// TIA Portal V16 export
// export: Created 2021-09-08T12:46:09.8350938Z, ExportSetting WithDefaults, DisplayName Totally Integrated Automation Portal, DisplayVersion V16 Update 3, DisplayName TIA Portal Version Control Interface, DisplayVersion V16 Update 2, DisplayName TIA Portal Openness, DisplayVersion V16 Update 3, DisplayName TIA Portal Teamcenter Gateway, DisplayVersion V16, DisplayName STEP 7 Professional, DisplayVersion V16 Update 3, DisplayName STEP 7 Safety, DisplayVersion V16, DisplayName WinCC Advanced, DisplayVersion V16 Update 3
FUNCTION_BLOCK "AvCntrl"   // FB81, LAD
{ S7_Optimized_Access := 'FALSE' }
VERSION : 0.1
// #ST:
// 0 0 - закрыта - стоп 
// 1 1- открыта - работа
// 2 2 -открывается - запускается
// 3 4 -закрывается - останавливается 
// 4 8 - ошибка питания
// 5 16 - ошибка концевиков - закрытия
// 6 32 - Блокировка
// 7 64 - сборная авария
// 8 128 - ошибка концевиков - открытия
// 9 256 - не выбран режим
// 10 - 512 - показывать кнопки ручного управления
// 
// БИТ 13 - РЕЖИМ
// бит 14 - состояние концевиков - открыто
// 15 - закрыто
// stored: AutoNumber false, IsIECCheckEnabled true, SetENOAutomatically false, UDAEnableTagReadback false
   VAR_INPUT
      power : Bool;   // питание устройства
      open : Bool;   // Задвижка открыта
      close : Bool;   // Задвижка закрыта
   END_VAR
   VAR_OUTPUT
      qKm : Bool;   // Выход на управление механизмом 0-стоп, 1-пуск
   END_VAR
   VAR_IN_OUT
      dev : "Av";
   END_VAR
   VAR DB_SPECIFIC
      Ack : Bool;   // Сброс Аварий
      ErrorOC : Bool;   // Признак аварии по закрытию или открытию
      ErrorPower : Bool;   // Признак аварии питания
      ErrorDis : Bool;   // Признак внешней блокировки
      Error : Bool;   // Признак наличия сборной ошибки
      qON : Bool;   // Выход для управления механизмом
      closed : Bool;
      opened : Bool;
      closing : Bool;
      opening : Bool;
      errOpen : Bool;
      errClose : Bool;
      timerOpening { S7_SetPoint := 'True'} : TON_TIME;
      timerClosing { S7_SetPoint := 'True'} : TON_TIME;
      tClose : Time;
      tOpen : Time;
   END_VAR
   VAR
      AvAckAlarm_Instance { S7_SetPoint := 'True'} : "AvAckAlarm";
   END_VAR
   VAR_TEMP
      tmpDInt : DInt;
   END_VAR
   VAR_TEMP   // added for the SCL form of the ladder/FBD networks
      _w1 : Bool;
   END_VAR
BEGIN

REGION Network 1: Сброс состояния
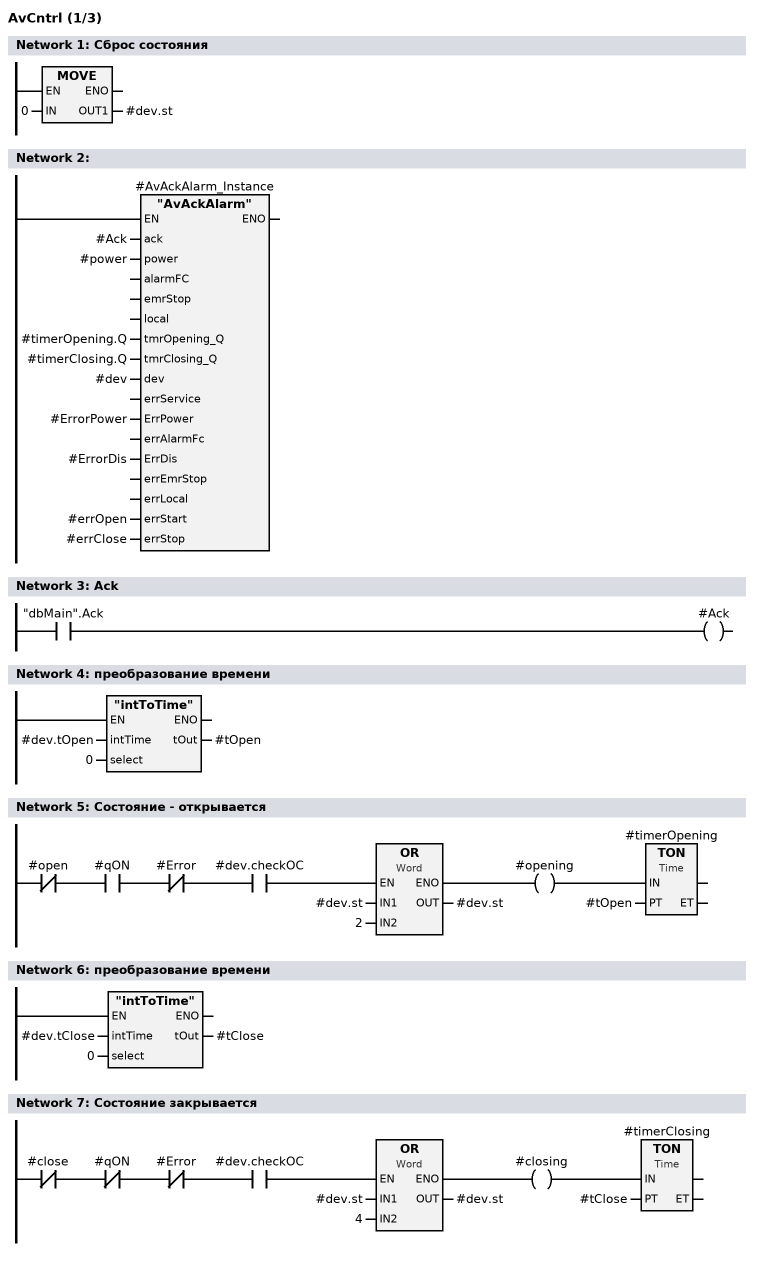
   RUNG wire#powerrail
      { S7_GenerateENO := "TRUE" } Move(in := 0, out1 => #dev.st)
   END_RUNG
   // the same network as SCL:
   #dev.st := 0;
END_REGION

REGION Network 2
   RUNG wire#powerrail
      #AvAckAlarm_Instance(ack := #Ack, power := #power, alarmFC :=, emrStop :=, local :=, tmrOpening_Q := #timerOpening.Q, tmrClosing_Q := #timerClosing.Q, dev := #dev, errService :=, ErrPower := #ErrorPower, errAlarmFc :=, ErrDis := #ErrorDis, errEmrStop :=, errLocal :=, errStart := #errOpen, errStop := #errClose)
   END_RUNG
   // the same network as SCL:
   #AvAckAlarm_Instance(ack := #Ack,   // "AvAckAlarm"
                        power := #power,
                        tmrOpening_Q := #timerOpening.Q,
                        tmrClosing_Q := #timerClosing.Q,
                        dev := #dev,
                        ErrPower := #ErrorPower,
                        ErrDis := #ErrorDis,
                        errStart := #errOpen,
                        errStop := #errClose);
END_REGION

REGION Network 3: Ack
   RUNG wire#powerrail
      Contact( "dbMain".Ack )
      Coil( #Ack )
   END_RUNG
   // the same network as SCL:
   #Ack := "dbMain".Ack;
END_REGION

REGION Network 4: преобразование времени
   RUNG wire#powerrail
      "intToTime"(intTime := #dev.tOpen, select := 0, tOut => #tOpen)
   END_RUNG
   // the same network as SCL:
   "intToTime"(intTime := #dev.tOpen, select := 0, tOut => #tOpen);
END_REGION

REGION Network 5: Состояние - открывается
   #_w1 := NOT #open AND #qON AND NOT #Error AND #dev.checkOC;
   IF #_w1 THEN #dev.st := #dev.st OR 2; END_IF;
   #opening := #_w1;
   #timerOpening(IN := #_w1, PT := #tOpen);   // TON
END_REGION

REGION Network 6: преобразование времени
   RUNG wire#powerrail
      "intToTime"(intTime := #dev.tClose, select := 0, tOut => #tClose)
   END_RUNG
   // the same network as SCL:
   "intToTime"(intTime := #dev.tClose, select := 0, tOut => #tClose);
END_REGION

REGION Network 7: Состояние закрывается
   #_w1 := NOT #close AND NOT #qON AND NOT #Error AND #dev.checkOC;
   IF #_w1 THEN #dev.st := #dev.st OR 4; END_IF;
   #closing := #_w1;
   #timerClosing(IN := #_w1, PT := #tClose);   // TON
END_REGION

REGION Network 8: Признак аварии по закрытию или открытию
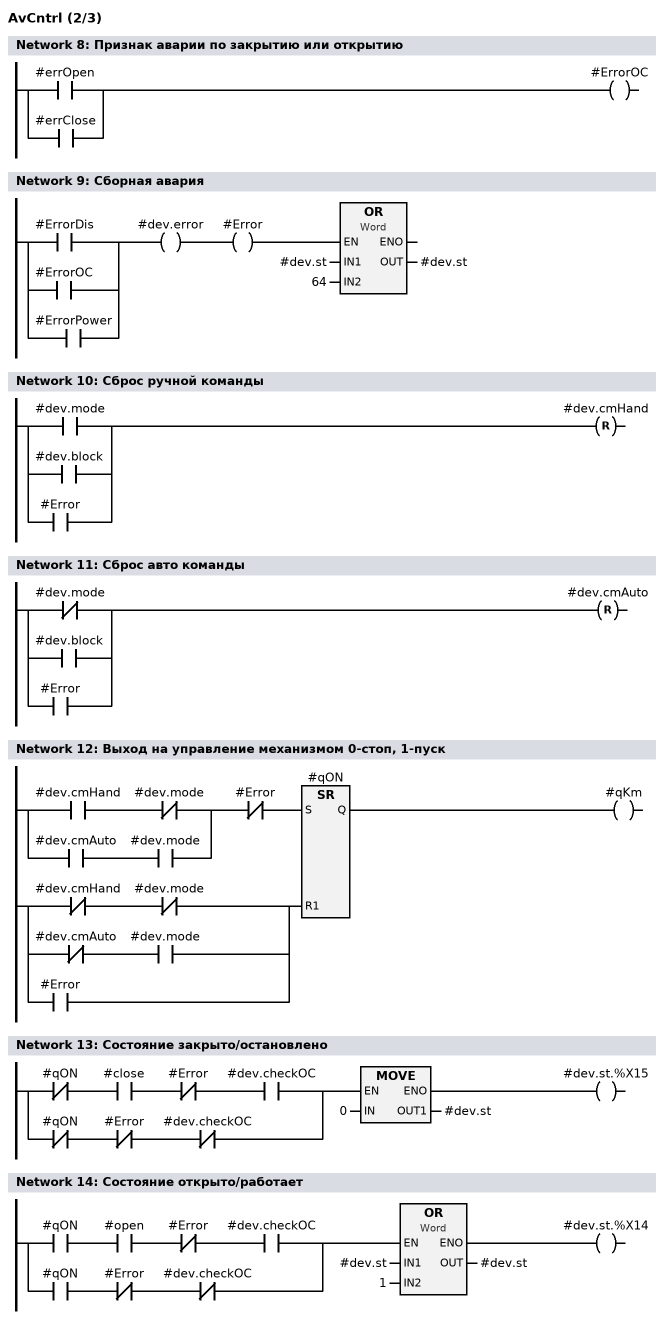
   RUNG wire#powerrail
      Contact( #errOpen )
      wire#w1
      Coil( #ErrorOC )
   END_RUNG
   RUNG wire#powerrail
      Contact( #errClose )
   END_RUNG wire#w1
   // the same network as SCL:
   #ErrorOC := #errOpen OR #errClose;
END_REGION

REGION Network 9: Сборная авария
   #dev.error := #ErrorDis OR #ErrorOC OR #ErrorPower;
   #Error := #dev.error;
   IF #dev.error THEN #dev.st := #dev.st OR 64; END_IF;
END_REGION

REGION Network 10: Сброс ручной команды
   RUNG wire#powerrail
      Contact( #dev.mode )
      wire#w1
      R_Coil( #dev.cmHand )
   END_RUNG
   RUNG wire#powerrail
      Contact( #dev.block )
   END_RUNG wire#w1
   RUNG wire#powerrail
      Contact( #Error )
   END_RUNG wire#w1
   // the same network as SCL:
   IF #dev.mode OR #dev.block OR #Error THEN #dev.cmHand := FALSE; END_IF;
END_REGION

REGION Network 11: Сброс авто команды
   RUNG wire#powerrail
      I_Contact( #dev.mode )
      wire#w1
      R_Coil( #dev.cmAuto )
   END_RUNG
   RUNG wire#powerrail
      Contact( #dev.block )
   END_RUNG wire#w1
   RUNG wire#powerrail
      Contact( #Error )
   END_RUNG wire#w1
   // the same network as SCL:
   IF NOT #dev.mode OR #dev.block OR #Error THEN #dev.cmAuto := FALSE; END_IF;
END_REGION

REGION Network 12: Выход на управление механизмом 0-стоп, 1-пуск
   RUNG wire#powerrail
      Contact( #dev.cmHand )
      I_Contact( #dev.mode )
      wire#w1
      I_Contact( #Error )
      S_SR(operand := #qON, r1 := wire#w2)
      Coil( #qKm )
   END_RUNG
   RUNG wire#powerrail
      Contact( #dev.cmAuto )
      Contact( #dev.mode )
   END_RUNG wire#w1
   RUNG wire#powerrail
      I_Contact( #dev.cmHand )
      I_Contact( #dev.mode )
   END_RUNG wire#w2
   RUNG wire#powerrail
      I_Contact( #dev.cmAuto )
      Contact( #dev.mode )
   END_RUNG wire#w2
   RUNG wire#powerrail
      Contact( #Error )
   END_RUNG wire#w2
   // the same network as SCL:
   IF ((#dev.cmHand AND NOT #dev.mode) OR (#dev.cmAuto AND #dev.mode)) AND NOT #Error THEN
       #qON := TRUE;   // SR flip-flop
   END_IF;
   IF (NOT #dev.cmHand AND NOT #dev.mode) OR (NOT #dev.cmAuto AND #dev.mode) OR #Error THEN
       #qON := FALSE;
   END_IF;
   #qKm := #qON;
END_REGION

REGION Network 13: Состояние закрыто/остановлено
   RUNG wire#powerrail
      I_Contact( #qON )
      Contact( #close )
      I_Contact( #Error )
      Contact( #dev.checkOC )
      wire#w1
      { S7_GenerateENO := "TRUE" } Move(in := 0, out1 => #dev.st)
      Coil( #dev.st.%X15 )
   END_RUNG
   RUNG wire#powerrail
      I_Contact( #qON )
      I_Contact( #Error )
      I_Contact( #dev.checkOC )
   END_RUNG wire#w1
   // the same network as SCL:
   // ENO of a box is taken as its EN; it also drops when the box reports an error
   #_w1 := (NOT #qON AND #close AND NOT #Error AND #dev.checkOC) OR (NOT #qON AND NOT #Error AND NOT #dev.checkOC);
   IF #_w1 THEN #dev.st := 0; END_IF;
   #dev.st.%X15 := #_w1;
END_REGION

REGION Network 14: Состояние открыто/работает
   #_w1 := (#qON AND #open AND NOT #Error AND #dev.checkOC) OR (#qON AND NOT #Error AND NOT #dev.checkOC);
   IF #_w1 THEN #dev.st := #dev.st OR 1; END_IF;
   #dev.st.%X14 := #_w1;
END_REGION

REGION Network 15: рУЧНОЙ режим для состояния
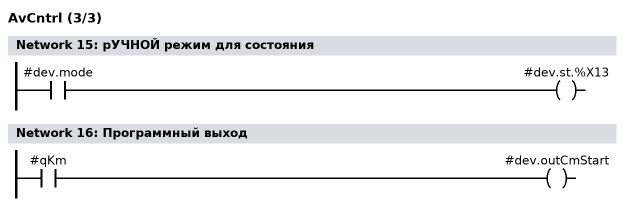
   RUNG wire#powerrail
      Contact( #dev.mode )
      Coil( #dev.st.%X13 )
   END_RUNG
   // the same network as SCL:
   #dev.st.%X13 := #dev.mode;
END_REGION

REGION Network 16: Программный выход
   RUNG wire#powerrail
      Contact( #qKm )
      Coil( #dev.outCmStart )
   END_RUNG
   // the same network as SCL:
   #dev.outCmStart := #qKm;
END_REGION
END_FUNCTION_BLOCK
